FUNCTION_BLOCK SludgeBufferLogic_2_HMI (* Service Interface Function Block Type *)
  (* Standard: 61499-2 *)
  (* Version 0.0, 10/24/2023, SESA685388, Schneider Electric, template *)
  PACKAGE SE.Nereda;
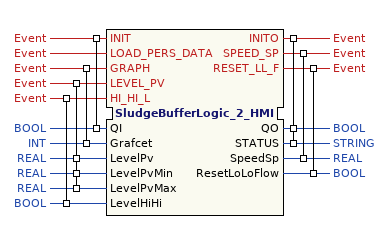
  EVENT_INPUT
    INIT WITH QI;
    LOAD_PERS_DATA;
    GRAPH WITH Grafcet;
    LEVEL_PV WITH LevelPv, LevelPvMin, LevelPvMax;
    HI_HI_L WITH LevelHiHi;
  END_EVENT
  EVENT_OUTPUT
    INITO WITH QO, STATUS;
    SPEED_SP WITH SpeedSp;
    RESET_LL_F WITH ResetLoLoFlow;
  END_EVENT
  VAR_INPUT
    QI : BOOL;
    Grafcet : INT;
    LevelPv : REAL;
    LevelPvMin : REAL;
    LevelPvMax : REAL;
    LevelHiHi : BOOL;
  END_VAR
  VAR_OUTPUT
    QO : BOOL; (* Event Output Qualifier *)
    STATUS : STRING; (* Service Status *)
    SpeedSp : REAL;
    ResetLoLoFlow : BOOL;
  END_VAR
  SERVICE /
    SEQUENCE 
    END_SEQUENCE
  END_SERVICE
END_FUNCTION_BLOCK
